// TIA Portal project "Report 1-5" (V15.1)

(* hardware
DEVICE "S7300/ET200M station_1"  S7-300 station
   slot 0: "Rail_0"  Rail  6ES7 390-1***0-0AA0
   slot 2: "PLC_1"  CPU 313C-2 DP  6ES7 313-6CF03-0AB0  V2.6
      slot 0: "MPI interface_1"  X1
      slot 1: "DP interface_1"  X2
      slot 2: "DI 16/DO 16_1"  DI16/DO16
      slot 4: "Count_1"  Counter
*)

// ===== PLC "PLC_1"  CPU 313C-2 DP =====

VAR_GLOBAL   // PLC tag table "Default tag table"
   "Start" AT %I0.0 : Bool;
   "Stop" AT %I0.1 : Bool;
   "Tag_1" AT %M0.0 : Bool;
   "Start_All" AT %M0.1 : Bool;
   "Tag_2" AT %M0.2 : Bool;
   "X1 Level" AT %I0.2 : Bool;
   "A Level" AT %Q0.0 : Bool;
   "X2 Level" AT %I0.3 : Bool;
   "Tag_3" AT %M0.3 : Bool;
   "B Level" AT %Q0.1 : Bool;
   "Timer 1" AT %T0 : Timer;
   "Blender" AT %Q0.2 : Bool;
   "Tag_4" AT %T1 : Timer;
   "Output" AT %Q0.3 : Bool;
END_VAR

ORGANIZATION_BLOCK "Main"   // OB1, LAD
TITLE = "Main Program Sweep (Cycle)"
{ S7_Optimized_Access := 'FALSE' }
VERSION : 0.1
   VAR_TEMP
      OB1_EV_CLASS : Byte;   // Bits 0-3 = 1 (Coming event), Bits 4-7 = 1 (Event class 1)
      OB1_SCAN_1 : Byte;   // 1 (Cold restart scan 1 of OB 1), 3 (Scan 2-n of OB 1)
      OB1_PRIORITY : Byte;   // Priority of OB Execution
      OB1_OB_NUMBR : Byte;   // 1 (Organization block 1, OB1)
      OB1_RESERVED_1 : Byte;   // Reserved for system
      OB1_RESERVED_2 : Byte;   // Reserved for system
      OB1_PREV_CYCLE : Int;   // Cycle time of previous OB1 scan (milliseconds)
      OB1_MIN_CYCLE : Int;   // Minimum cycle time of OB1 (milliseconds)
      OB1_MAX_CYCLE : Int;   // Maximum cycle time of OB1 (milliseconds)
      OB1_DATE_TIME : Date_And_Time;   // Date and time OB1 started
   END_VAR
   VAR_TEMP   // added for the SCL form of the ladder/FBD networks
      _w1 : Bool;
      _s5time1 : S5Time;
   END_VAR
BEGIN

REGION Network 1
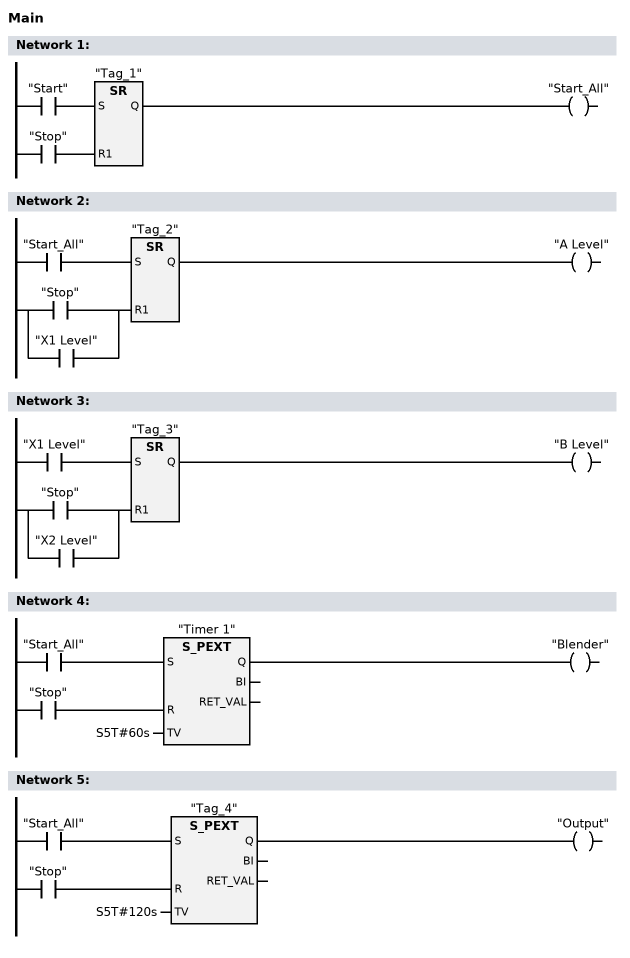
   RUNG wire#powerrail
      Contact( "Start" )
      S_SR(operand := "Tag_1", r1 := wire#w1)
      Coil( "Start_All" )
   END_RUNG
   RUNG wire#powerrail
      Contact( "Stop" )
   END_RUNG wire#w1
   // the same network as SCL:
   IF "Start" THEN
       "Tag_1" := TRUE;   // SR flip-flop
   END_IF;
   IF "Stop" THEN "Tag_1" := FALSE; END_IF;
   "Start_All" := "Tag_1";
END_REGION

REGION Network 2
   RUNG wire#powerrail
      Contact( "Start_All" )
      S_SR(operand := "Tag_2", r1 := wire#w1)
      Coil( "A Level" )
   END_RUNG
   RUNG wire#powerrail
      Contact( "Stop" )
   END_RUNG wire#w1
   RUNG wire#powerrail
      Contact( "X1 Level" )
   END_RUNG wire#w1
   // the same network as SCL:
   IF "Start_All" THEN
       "Tag_2" := TRUE;   // SR flip-flop
   END_IF;
   IF "Stop" OR "X1 Level" THEN "Tag_2" := FALSE; END_IF;
   "A Level" := "Tag_2";
END_REGION

REGION Network 3
   RUNG wire#powerrail
      Contact( "X1 Level" )
      S_SR(operand := "Tag_3", r1 := wire#w1)
      Coil( "B Level" )
   END_RUNG
   RUNG wire#powerrail
      Contact( "Stop" )
   END_RUNG wire#w1
   RUNG wire#powerrail
      Contact( "X2 Level" )
   END_RUNG wire#w1
   // the same network as SCL:
   IF "X1 Level" THEN
       "Tag_3" := TRUE;   // SR flip-flop
   END_IF;
   IF "Stop" OR "X2 Level" THEN "Tag_3" := FALSE; END_IF;
   "B Level" := "Tag_3";
END_REGION

REGION Network 4
   RUNG wire#powerrail
      Contact( "Start_All" )
      S_PEXT(T_NO := "Timer 1", R := wire#w1, TV := S5T#60s, BI =>, RET_VAL =>)
      Coil( "Blender" )
   END_RUNG
   RUNG wire#powerrail
      Contact( "Stop" )
   END_RUNG wire#w1
   // the same network as SCL:
   #_s5time1 := S_PEXT(T_NO := "Timer 1", S := "Start_All", R := "Stop", TV := S5T#60s, Q => #_w1);
   "Blender" := #_w1;
END_REGION

REGION Network 5
   RUNG wire#powerrail
      Contact( "Start_All" )
      S_PEXT(T_NO := "Tag_4", R := wire#w1, TV := S5T#120s, BI =>, RET_VAL =>)
      Coil( "Output" )
   END_RUNG
   RUNG wire#powerrail
      Contact( "Stop" )
   END_RUNG wire#w1
   // the same network as SCL:
   #_s5time1 := S_PEXT(T_NO := "Tag_4", S := "Start_All", R := "Stop", TV := S5T#120s, Q => #_w1);
   "Output" := #_w1;
END_REGION
END_ORGANIZATION_BLOCK